(* CODESYS project Singla_Jagdamba_Rice_Final_28_02_20.project
   Title: Singla_Jagdamba_Rice_23_09_18
   Version: 0.0.0.0

Project tree, tasks and I/O mapping:
  MyController : TM218LDA40DRN, Schneider Electric, order no. TM218LDA40DRN, version 4.0.1.26
    application Application
      task MAST (cyclic, interval 20 ms, priority 15, watchdog 100 ms x 1) calls MainPOU
      function HiddenPOU [ST]
      global variables GVL
      program MainPOU [LD]
      function block fx1 [ST]
      function block fx2 [ST]
      function block CylOpenClose [ST]
    Embedded Functions
      IO : IO, Schneider Electric, version 4.0.1.26
          input  ES1 : BOOL  // ID0.I0
          input  ES2 : BOOL  // ID0.I1
          input  ES3 : BOOL  // ID0.I2
          input  ES4 : BOOL  // ID0.I3
          input  ES5 : BOOL  // ID0.I4
          input  ES6 : BOOL  // ID0.I5
          input  ES7 : BOOL  // ID0.I6
          input  ES8 : BOOL  // ID0.I7
          input  PS1 : BOOL  // ID0.I8
          input  PS2 : BOOL  // ID0.I9
          input  PS3 : BOOL  // ID0.I10
          input  PS4 : BOOL  // ID0.I11
          input  PS5 : BOOL  // ID0.I12
          input  PS6 : BOOL  // ID0.I13
          input  PS7 : BOOL  // ID0.I14
          input  PS8 : BOOL  // ID0.I15
          output qCylinder1 : BOOL  // QW0.Q0
          output qCylinder2 : BOOL  // QW0.Q1
          output qCylinder3 : BOOL  // QW0.Q2
          output qCylinder4 : BOOL  // QW0.Q3
          output qCylinder5 : BOOL  // QW0.Q4
          output qCylinder6 : BOOL  // QW0.Q5
          output qCylinder7 : BOOL  // QW0.Q6
          output qCylinder8 : BOOL  // QW0.Q7
          output qCylinder9 : BOOL  // QW0.Q8
          output qCylinder10 : BOOL  // QW0.Q9
          output qCylinder11 : BOOL  // QW0.Q10
          output qCylinder12 : BOOL  // QW0.Q11
          output qCylinder13 : BOOL  // QW0.Q12
          output qCylinder14 : BOOL  // QW0.Q13
          unmapped channels: ID0, QW0
      HSC : HSC, Schneider Electric, version 4.0.1.26
    Serial Line 1
      SoMachine_Network_Manager : SoMachine-Network Manager, Schneider Electric, version 4.0.0.2
    Serial Line 2
      Modbus_Manager : Modbus Manager, Schneider Electric, version 4.0.0.2
*)

// MyController/Application/GVL
VAR_GLOBAL
	
	k1TopCylClose: BOOL;
	k2TopCylClose: BOOL;
	k3TopCylClose: BOOL;
	k4TopCylClose: BOOL;
	k5TopCylClose: BOOL;
	k6TopCylClose: BOOL;
	
	manualOpenCyl1 AT %MX608.0: BOOL;
	manualOpenCyl2 AT %MX608.1: BOOL;
	manualOpenCyl3 AT %MX608.2: BOOL;
	manualOpenCyl4 AT %MX608.3: BOOL;
	manualOpenCyl5 AT %MX608.4: BOOL;
	manualOpenCyl6 AT %MX608.5: BOOL;
	manualOpenCyl7 AT %MX608.6: BOOL;
	manualOpenCyl8 AT %MX608.7: BOOL;
	manualOpenCyl9 AT %MX609.0: BOOL;
	manualOpenCyl10 AT %MX609.1: BOOL;
	manualOpenCyl11 AT %MX617.0: BOOL;
	manualOpenCyl12 AT %MX617.1: BOOL;
	manualOpenCyl13 AT %MX617.2: BOOL;
	manualOpenCyl14 AT %MX617.3: BOOL;
	
	manualCloseCyl1 AT %MX609.2: BOOL;
	manualCloseCyl2 AT %MX609.3: BOOL;
	manualCloseCyl3 AT %MX609.4: BOOL;
	manualCloseCyl4 AT %MX609.5: BOOL;
	manualCloseCyl5 AT %MX609.6: BOOL;
	manualCloseCyl6 AT %MX609.7: BOOL;
	manualCloseCyl7 AT %MX610.0: BOOL;
	manualCloseCyl8 AT %MX610.1: BOOL;
	manualCloseCyl9 AT %MX610.2: BOOL;
	manualCloseCyl10 AT %MX610.3: BOOL;
	manualCloseCyl11 AT %MX617.4: BOOL;
	manualCloseCyl12 AT %MX617.5: BOOL;
	manualCloseCyl13 AT %MX617.6: BOOL;
	manualCloseCyl14 AT %MX617.7: BOOL;
	
	
	openCyl1 AT %MX603.2: BOOL;
	openCyl2 AT %MX603.3: BOOL;
	openCyl3 AT %MX603.4: BOOL;
	openCyl4 AT %MX603.5: BOOL;
	openCyl5 AT %MX603.6: BOOL;
	openCyl6 AT %MX603.7: BOOL;
	openCyl7 AT %MX604.0: BOOL;
	openCyl8 AT %MX604.1: BOOL;
	openCyl9 AT %MX604.2: BOOL;
	openCyl10 AT %MX604.3: BOOL;
	openCyl11 AT %MX618.0: BOOL;
	openCyl12 AT %MX618.1: BOOL;
	openCyl13 AT %MX618.2: BOOL;
	openCyl14 AT %MX618.3: BOOL;
	
	k1CycleStart AT %MX606.0: BOOL;
	k2CycleStart AT %MX606.1: BOOL;
	k3CycleStart AT %MX606.2: BOOL;
	k4CycleStart AT %MX606.3: BOOL;
	k5CycleStart AT %MX618.4: BOOL;
	k6CycleStart AT %MX618.5: BOOL;
	p1CycleStart AT %MX606.4: BOOL;
	p2CycleStart AT %MX606.5: BOOL;
	
	k1CycleStop AT %MX606.6: BOOL;
	k2CycleStop AT %MX606.7: BOOL;
	k3CycleStop AT %MX607.0: BOOL;
	k4CycleStop AT %MX607.1: BOOL;
	k5CycleStop AT %MX618.6: BOOL;
	k6CycleStop AT %MX618.7: BOOL;
	p1CycleStop AT %MX607.2: BOOL;
	p2CycleStop AT %MX607.3: BOOL;
	
	k1Start AT %MX612.0: BOOL;
	k2Start AT %MX612.1: BOOL;
	k3Start AT %MX612.2: BOOL;
	k4Start AT %MX612.3: BOOL;
	k5Start AT %MX619.0: BOOL;
	k6Start AT %MX619.1: BOOL;
	p1Start AT %MX612.4: BOOL;
	p2Start AT %MX612.5: BOOL;

	k1CountComplete AT %MX612.6: BOOL;
	k2CountComplete AT %MX612.7: BOOL;
	k3CountComplete AT %MX613.0: BOOL;
	k4CountComplete AT %MX613.1: BOOL;
	k5CountComplete AT %MX619.2: BOOL;
	k6CountComplete AT %MX619.3: BOOL;
	p1CountComplete AT %MX613.2: BOOL;
	p2CountComplete AT %MX613.3: BOOL;
	
	k1PressureLow AT %MX613.4: BOOL;
	k2PressureLow AT %MX613.5: BOOL;
	k3PressureLow AT %MX613.6: BOOL;
	k4PressureLow AT %MX613.7: BOOL;
	k5PressureLow AT %MX619.4: BOOL;
	k6PressureLow AT %MX619.5: BOOL;
	p1PressureLow AT %MX614.0: BOOL;
	p2PressureLow AT %MX614.1: BOOL;
	
	k1Reset AT %MX616.0: BOOL;
	k2Reset AT %MX616.1: BOOL;
	k3Reset AT %MX616.2: BOOL;
	k4Reset AT %MX616.3: BOOL;
	k5Reset AT %MX619.6: BOOL;
	k6Reset AT %MX619.7: BOOL;
	p1Reset AT %MX616.4: BOOL;
	p2Reset AT %MX616.5: BOOL;
	
	k1ActCycleTime AT %MW122: INT; //in minutes
	k2ActCycleTime AT %MW123: INT;
	k3ActCycleTime AT %MW124: INT;
	k4ActCycleTime AT %MW125: INT;
	k5ActCycleTime AT %MW152: INT;
	k6ActCycleTime AT %MW153: INT;
	p1ActCycleTime AT %MW126: INT;
	p2ActCycleTime AT %MW127: INT;
	
	k1ActCount AT %MW128: INT;
	k2ActCount AT %MW129: INT;
	k3ActCount AT %MW130: INT;
	k4ActCount AT %MW131: INT;
	k5ActCount AT %MW150: INT;
	k6ActCount AT %MW151: INT;
	p1ActCount AT %MW132: INT;
	p2ActCount AT %MW133: INT;
	
END_VAR

VAR_GLOBAL RETAIN
	k1SetCount AT %MW100: INT := 15;
	k2SetCount AT %MW101: INT := 15;
	k3SetCount AT %MW102: INT := 15;
	k4SetCount AT %MW103: INT := 15;
	k5SetCount AT %MW148: INT := 15;
	k6SetCount AT %MW149: INT := 15;
	p1SetCount AT %MW104: INT := 5;
	p2SetCount AT %MW105: INT := 5;
	
	setTimeCylOpen1 AT %MW106: INT := 15; //in seconds
	setTimeCylOpen2 AT %MW107: INT := 15;
	setTimeCylOpen3 AT %MW108: INT := 15;
	setTimeCylOpen4 AT %MW109: INT := 15;
	setTimeCylOpen5 AT %MW110: INT := 15;
	setTimeCylOpen6 AT %MW111: INT := 15;
	setTimeCylOpen7 AT %MW112: INT := 15;
	setTimeCylOpen8 AT %MW113: INT := 15;
	setTimeCylOpen9 AT %MW114: INT := 15;
	setTimeCylOpen10 AT %MW115: INT := 15;
	setTimeCylOpen11 AT %MW144: INT := 15;
	setTimeCylOpen12 AT %MW145: INT := 15;
	setTimeCylOpen13 AT %MW146: INT := 15;
	setTimeCylOpen14 AT %MW147: INT := 15;
	
	
	k1SetCycleTime AT %MW116: INT := 15;
	k2SetCycleTime AT %MW117: INT := 15;
	k3SetCycleTime AT %MW118: INT := 15;
	k4SetCycleTime AT %MW119: INT := 15;
	k5SetCycleTime AT %MW142: INT := 15;
	k6SetCycleTime AT %MW143: INT := 15;
	p1SetCycleTime AT %MW120: INT := 15;
	p2SetCycleTime AT %MW121: INT := 15;
	
	k1SetCloseCount AT %MW134: INT := 2;
	k2SetCloseCount AT %MW135: INT := 2;
	k3SetCloseCount AT %MW136: INT := 2;
	k4SetCloseCount AT %MW137: INT := 2;
	k5SetCloseCount AT %MW140: INT := 2;
	k6SetCloseCount AT %MW141: INT := 2;
	p1SetCloseCount AT %MW138: INT;
	p2SetCloseCount AT %MW139: INT;
	
	k1ManualOverride AT %MX600.0: BOOL;
	k2ManualOverride AT %MX600.1: BOOL;
	k3ManualOverride AT %MX600.2: BOOL;
	k4ManualOverride AT %MX600.3: BOOL;
	k5ManualOverride AT %MX620.0: BOOL;
	k6ManualOverride AT %MX620.1: BOOL;
	p1ManualOverride AT %MX600.4: BOOL;
	p2ManualOverride AT %MX600.5: BOOL;

END_VAR

// MyController/Application/MainPOU
PROGRAM MainPOU
VAR

	Kacchi_1: fx1;
	Kacchi_1_Count: fx2;
	Kacchi_2: fx1;
	Kacchi_2_Count: fx2;
	Kacchi_3_Count: fx2;
	Kacchi_3: fx1;
	Kacchi_4: fx1;
	Kacchi_4_Count: fx2;
	Pakki_1: fx1;
	Pakki_1_Count: fx2;
	Pakki_2: fx1;
	Pakki_2_Count: fx2;
	
	
	k2BottomCmd: BOOL;
	k1BottomCmd: BOOL;
	k3BottomCmd: BOOL;
	k4BottomCmd: BOOL;
	p1BottomCmd: BOOL;
	p2BottomCmd: BOOL;
	
	CylOpenClose_0: CylOpenClose;
	CylOpenClose_1: CylOpenClose;
	CylOpenClose_2: CylOpenClose;
	CylOpenClose_3: CylOpenClose;
	CylOpenClose_4: CylOpenClose;
	CylOpenClose_5: CylOpenClose;
	CylOpenClose_6: CylOpenClose;
	CylOpenClose_7: CylOpenClose;
	CylOpenClose_8: CylOpenClose;
	CylOpenClose_9: CylOpenClose;
	p2Stop: BOOL;
	k4Stop: BOOL;
	p1Stop: BOOL;
	k3Stop: BOOL;
	k2Stop: BOOL;
	k1Stop: BOOL;
	
	R_TRIG_0: R_TRIG;
	R_TRIG_1: R_TRIG;
	R_TRIG_2: R_TRIG;
	R_TRIG_3: R_TRIG;
	R_TRIG_4: R_TRIG;
	R_TRIG_5: R_TRIG;
	R_TRIG_6: R_TRIG;
	R_TRIG_7: R_TRIG;
	R_TRIG_8: R_TRIG;
	R_TRIG_9: R_TRIG;
	RS_6: RS;
	k6Stop: BOOL;
	R_TRIG_15: R_TRIG;
	R_TRIG_16: R_TRIG;
	RS_7: RS;
	Kacchi_5: fx1;
	k5BottomCmd: BOOL;
	Kacchi_5_Count: fx2;
	k5Stop: BOOL;
	Kacchi_6: fx1;
	k6BottomCmd: BOOL;
	Kacchi_6_Count: fx2;
	CylOpenClose_10: CylOpenClose;
	R_TRIG_10: R_TRIG;
	CylOpenClose_11: CylOpenClose;
	CylOpenClose_12: CylOpenClose;
	R_TRIG_12: R_TRIG;
	CylOpenClose_13: CylOpenClose;
END_VAR

VAR RETAIN
	RS_0: RS;
	RS_1: RS;
	RS_2: RS;
	RS_3: RS;
	RS_4: RS;
	RS_5: RS;
END_VAR
VAR // added by the converter: edge detectors and wires of the graphical bodies
    _w1, _w2 : BOOL;
END_VAR

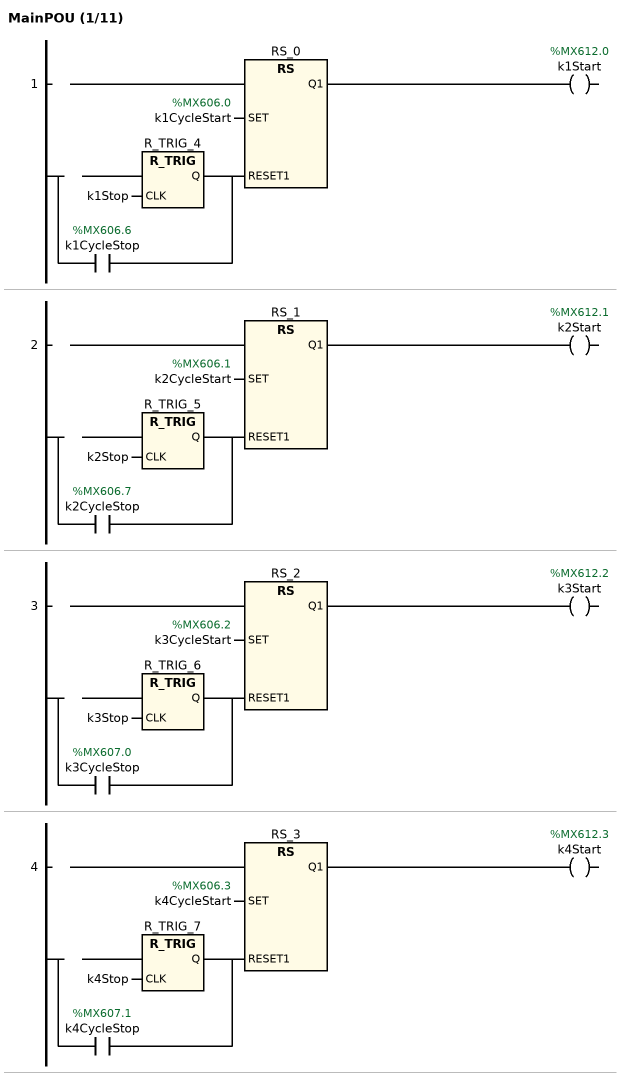
// NETWORK 1
//   k1CycleStart: AT %MX606.0
//   k1CycleStop: AT %MX606.6
//   k1Start: AT %MX612.0
R_TRIG_4(CLK := k1Stop); // R_TRIG
RS_0(SET := k1CycleStart, RESET1 := R_TRIG_4.Q OR k1CycleStop); // RS
k1Start := RS_0.Q1;

// NETWORK 2
//   k2CycleStart: AT %MX606.1
//   k2CycleStop: AT %MX606.7
//   k2Start: AT %MX612.1
R_TRIG_5(CLK := k2Stop); // R_TRIG
RS_1(SET := k2CycleStart, RESET1 := R_TRIG_5.Q OR k2CycleStop); // RS
k2Start := RS_1.Q1;

// NETWORK 3
//   k3CycleStart: AT %MX606.2
//   k3CycleStop: AT %MX607.0
//   k3Start: AT %MX612.2
R_TRIG_6(CLK := k3Stop); // R_TRIG
RS_2(SET := k3CycleStart, RESET1 := R_TRIG_6.Q OR k3CycleStop); // RS
k3Start := RS_2.Q1;

// NETWORK 4
//   k4CycleStart: AT %MX606.3
//   k4CycleStop: AT %MX607.1
//   k4Start: AT %MX612.3
R_TRIG_7(CLK := k4Stop); // R_TRIG
RS_3(SET := k4CycleStart, RESET1 := R_TRIG_7.Q OR k4CycleStop); // RS
k4Start := RS_3.Q1;

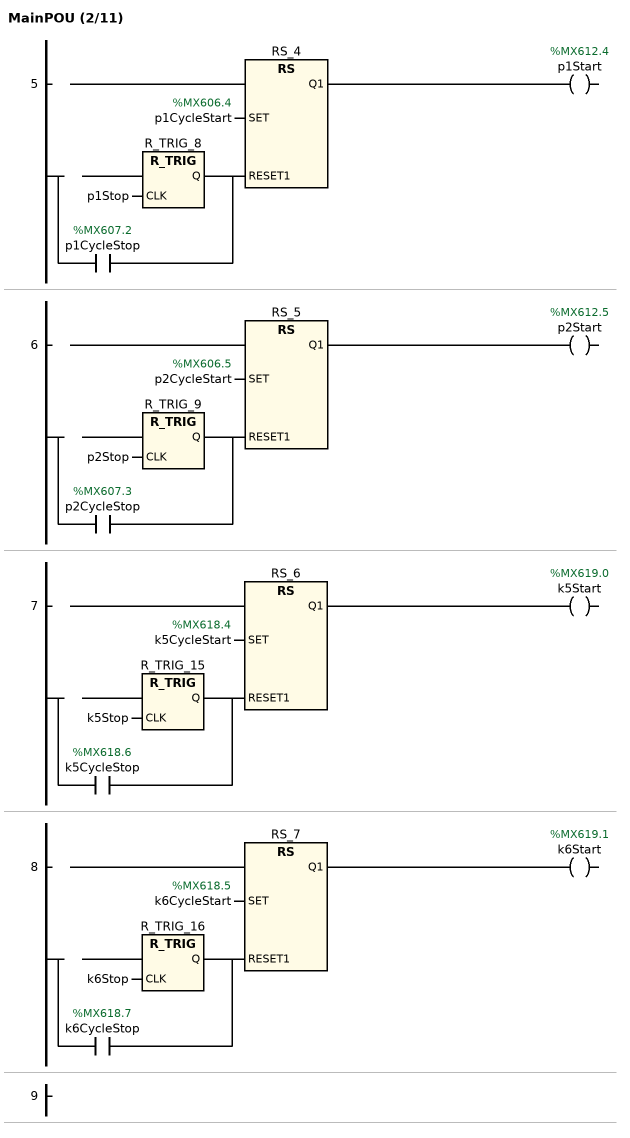
// NETWORK 5
//   p1CycleStart: AT %MX606.4
//   p1CycleStop: AT %MX607.2
//   p1Start: AT %MX612.4
R_TRIG_8(CLK := p1Stop); // R_TRIG
RS_4(SET := p1CycleStart, RESET1 := R_TRIG_8.Q OR p1CycleStop); // RS
p1Start := RS_4.Q1;

// NETWORK 6
//   p2CycleStart: AT %MX606.5
//   p2CycleStop: AT %MX607.3
//   p2Start: AT %MX612.5
R_TRIG_9(CLK := p2Stop); // R_TRIG
RS_5(SET := p2CycleStart, RESET1 := R_TRIG_9.Q OR p2CycleStop); // RS
p2Start := RS_5.Q1;

// NETWORK 7
//   k5CycleStart: AT %MX618.4
//   k5CycleStop: AT %MX618.6
//   k5Start: AT %MX619.0
R_TRIG_15(CLK := k5Stop); // R_TRIG
RS_6(SET := k5CycleStart, RESET1 := R_TRIG_15.Q OR k5CycleStop); // RS
k5Start := RS_6.Q1;

// NETWORK 8
//   k6CycleStart: AT %MX618.5
//   k6CycleStop: AT %MX618.7
//   k6Start: AT %MX619.1
R_TRIG_16(CLK := k6Stop); // R_TRIG
RS_7(SET := k6CycleStart, RESET1 := R_TRIG_16.Q OR k6CycleStop); // RS
k6Start := RS_7.Q1;

// NETWORK 9

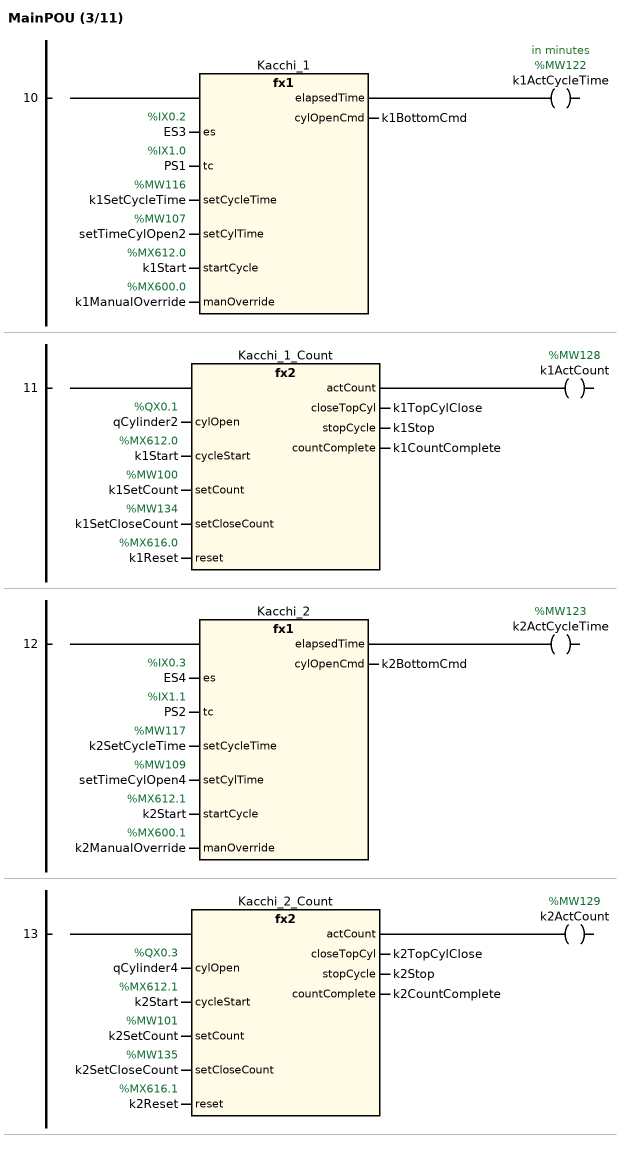
// NETWORK 10
//   ES3: IO : | AT %IX0.2
//   PS1: IO : | AT %IX1.0
//   k1SetCycleTime: AT %MW116
//   setTimeCylOpen2: AT %MW107
//   k1Start: AT %MX612.0
//   k1ManualOverride: AT %MX600.0
//   k1ActCycleTime: in minutes | AT %MW122
Kacchi_1(
    es := ES3,
    tc := PS1,
    setCycleTime := k1SetCycleTime,
    setCylTime := setTimeCylOpen2,
    startCycle := k1Start,
    manOverride := k1ManualOverride,
    cylOpenCmd => k1BottomCmd); // fx1
k1ActCycleTime := Kacchi_1.elapsedTime;

// NETWORK 11
//   qCylinder2: IO : | AT %QX0.1
//   k1Start: AT %MX612.0
//   k1SetCount: AT %MW100
//   k1SetCloseCount: AT %MW134
//   k1Reset: AT %MX616.0
//   k1CountComplete: AT %MX612.6
//   k1ActCount: AT %MW128
Kacchi_1_Count(
    cylOpen := qCylinder2,
    cycleStart := k1Start,
    setCount := k1SetCount,
    setCloseCount := k1SetCloseCount,
    reset := k1Reset,
    closeTopCyl => k1TopCylClose,
    stopCycle => k1Stop,
    countComplete => k1CountComplete); // fx2
k1ActCount := Kacchi_1_Count.actCount;

// NETWORK 12
//   ES4: IO : | AT %IX0.3
//   PS2: IO : | AT %IX1.1
//   k2SetCycleTime: AT %MW117
//   setTimeCylOpen4: AT %MW109
//   k2Start: AT %MX612.1
//   k2ManualOverride: AT %MX600.1
//   k2ActCycleTime: AT %MW123
Kacchi_2(
    es := ES4,
    tc := PS2,
    setCycleTime := k2SetCycleTime,
    setCylTime := setTimeCylOpen4,
    startCycle := k2Start,
    manOverride := k2ManualOverride,
    cylOpenCmd => k2BottomCmd); // fx1
k2ActCycleTime := Kacchi_2.elapsedTime;

// NETWORK 13
//   qCylinder4: IO : | AT %QX0.3
//   k2Start: AT %MX612.1
//   k2SetCount: AT %MW101
//   k2SetCloseCount: AT %MW135
//   k2Reset: AT %MX616.1
//   k2CountComplete: AT %MX612.7
//   k2ActCount: AT %MW129
Kacchi_2_Count(
    cylOpen := qCylinder4,
    cycleStart := k2Start,
    setCount := k2SetCount,
    setCloseCount := k2SetCloseCount,
    reset := k2Reset,
    closeTopCyl => k2TopCylClose,
    stopCycle => k2Stop,
    countComplete => k2CountComplete); // fx2
k2ActCount := Kacchi_2_Count.actCount;

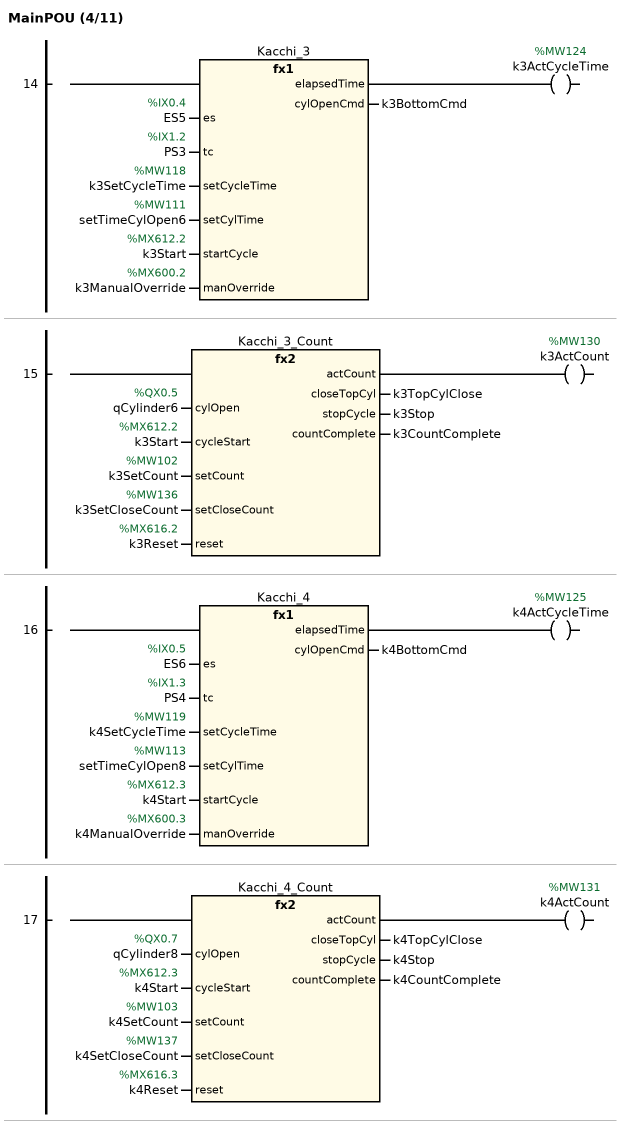
// NETWORK 14
//   ES5: IO : | AT %IX0.4
//   PS3: IO : | AT %IX1.2
//   k3SetCycleTime: AT %MW118
//   setTimeCylOpen6: AT %MW111
//   k3Start: AT %MX612.2
//   k3ManualOverride: AT %MX600.2
//   k3ActCycleTime: AT %MW124
Kacchi_3(
    es := ES5,
    tc := PS3,
    setCycleTime := k3SetCycleTime,
    setCylTime := setTimeCylOpen6,
    startCycle := k3Start,
    manOverride := k3ManualOverride,
    cylOpenCmd => k3BottomCmd); // fx1
k3ActCycleTime := Kacchi_3.elapsedTime;

// NETWORK 15
//   qCylinder6: IO : | AT %QX0.5
//   k3Start: AT %MX612.2
//   k3SetCount: AT %MW102
//   k3SetCloseCount: AT %MW136
//   k3Reset: AT %MX616.2
//   k3CountComplete: AT %MX613.0
//   k3ActCount: AT %MW130
Kacchi_3_Count(
    cylOpen := qCylinder6,
    cycleStart := k3Start,
    setCount := k3SetCount,
    setCloseCount := k3SetCloseCount,
    reset := k3Reset,
    closeTopCyl => k3TopCylClose,
    stopCycle => k3Stop,
    countComplete => k3CountComplete); // fx2
k3ActCount := Kacchi_3_Count.actCount;

// NETWORK 16
//   ES6: IO : | AT %IX0.5
//   PS4: IO : | AT %IX1.3
//   k4SetCycleTime: AT %MW119
//   setTimeCylOpen8: AT %MW113
//   k4Start: AT %MX612.3
//   k4ManualOverride: AT %MX600.3
//   k4ActCycleTime: AT %MW125
Kacchi_4(
    es := ES6,
    tc := PS4,
    setCycleTime := k4SetCycleTime,
    setCylTime := setTimeCylOpen8,
    startCycle := k4Start,
    manOverride := k4ManualOverride,
    cylOpenCmd => k4BottomCmd); // fx1
k4ActCycleTime := Kacchi_4.elapsedTime;

// NETWORK 17
//   qCylinder8: IO : | AT %QX0.7
//   k4Start: AT %MX612.3
//   k4SetCount: AT %MW103
//   k4SetCloseCount: AT %MW137
//   k4Reset: AT %MX616.3
//   k4CountComplete: AT %MX613.1
//   k4ActCount: AT %MW131
Kacchi_4_Count(
    cylOpen := qCylinder8,
    cycleStart := k4Start,
    setCount := k4SetCount,
    setCloseCount := k4SetCloseCount,
    reset := k4Reset,
    closeTopCyl => k4TopCylClose,
    stopCycle => k4Stop,
    countComplete => k4CountComplete); // fx2
k4ActCount := Kacchi_4_Count.actCount;

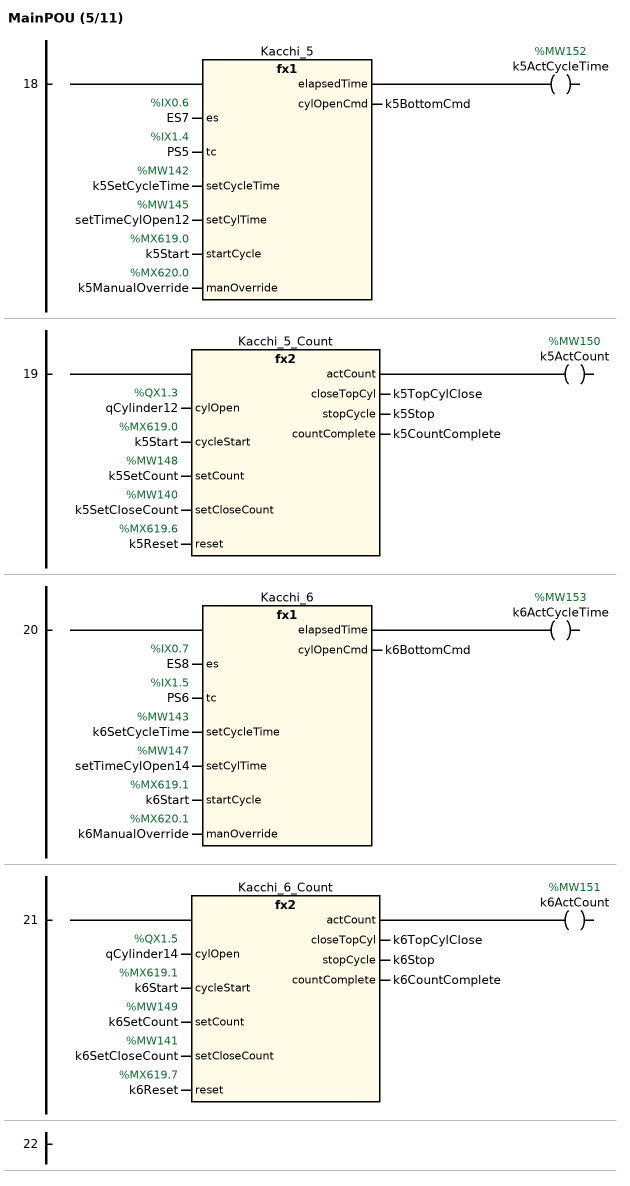
// NETWORK 18
//   ES7: IO : | AT %IX0.6
//   PS5: IO : | AT %IX1.4
//   k5SetCycleTime: AT %MW142
//   setTimeCylOpen12: AT %MW145
//   k5Start: AT %MX619.0
//   k5ManualOverride: AT %MX620.0
//   k5ActCycleTime: AT %MW152
Kacchi_5(
    es := ES7,
    tc := PS5,
    setCycleTime := k5SetCycleTime,
    setCylTime := setTimeCylOpen12,
    startCycle := k5Start,
    manOverride := k5ManualOverride,
    cylOpenCmd => k5BottomCmd); // fx1
k5ActCycleTime := Kacchi_5.elapsedTime;

// NETWORK 19
//   qCylinder12: IO : | AT %QX1.3
//   k5Start: AT %MX619.0
//   k5SetCount: AT %MW148
//   k5SetCloseCount: AT %MW140
//   k5Reset: AT %MX619.6
//   k5CountComplete: AT %MX619.2
//   k5ActCount: AT %MW150
Kacchi_5_Count(
    cylOpen := qCylinder12,
    cycleStart := k5Start,
    setCount := k5SetCount,
    setCloseCount := k5SetCloseCount,
    reset := k5Reset,
    closeTopCyl => k5TopCylClose,
    stopCycle => k5Stop,
    countComplete => k5CountComplete); // fx2
k5ActCount := Kacchi_5_Count.actCount;

// NETWORK 20
//   ES8: IO : | AT %IX0.7
//   PS6: IO : | AT %IX1.5
//   k6SetCycleTime: AT %MW143
//   setTimeCylOpen14: AT %MW147
//   k6Start: AT %MX619.1
//   k6ManualOverride: AT %MX620.1
//   k6ActCycleTime: AT %MW153
Kacchi_6(
    es := ES8,
    tc := PS6,
    setCycleTime := k6SetCycleTime,
    setCylTime := setTimeCylOpen14,
    startCycle := k6Start,
    manOverride := k6ManualOverride,
    cylOpenCmd => k6BottomCmd); // fx1
k6ActCycleTime := Kacchi_6.elapsedTime;

// NETWORK 21
//   qCylinder14: IO : | AT %QX1.5
//   k6Start: AT %MX619.1
//   k6SetCount: AT %MW149
//   k6SetCloseCount: AT %MW141
//   k6Reset: AT %MX619.7
//   k6CountComplete: AT %MX619.3
//   k6ActCount: AT %MW151
Kacchi_6_Count(
    cylOpen := qCylinder14,
    cycleStart := k6Start,
    setCount := k6SetCount,
    setCloseCount := k6SetCloseCount,
    reset := k6Reset,
    closeTopCyl => k6TopCylClose,
    stopCycle => k6Stop,
    countComplete => k6CountComplete); // fx2
k6ActCount := Kacchi_6_Count.actCount;

// NETWORK 22

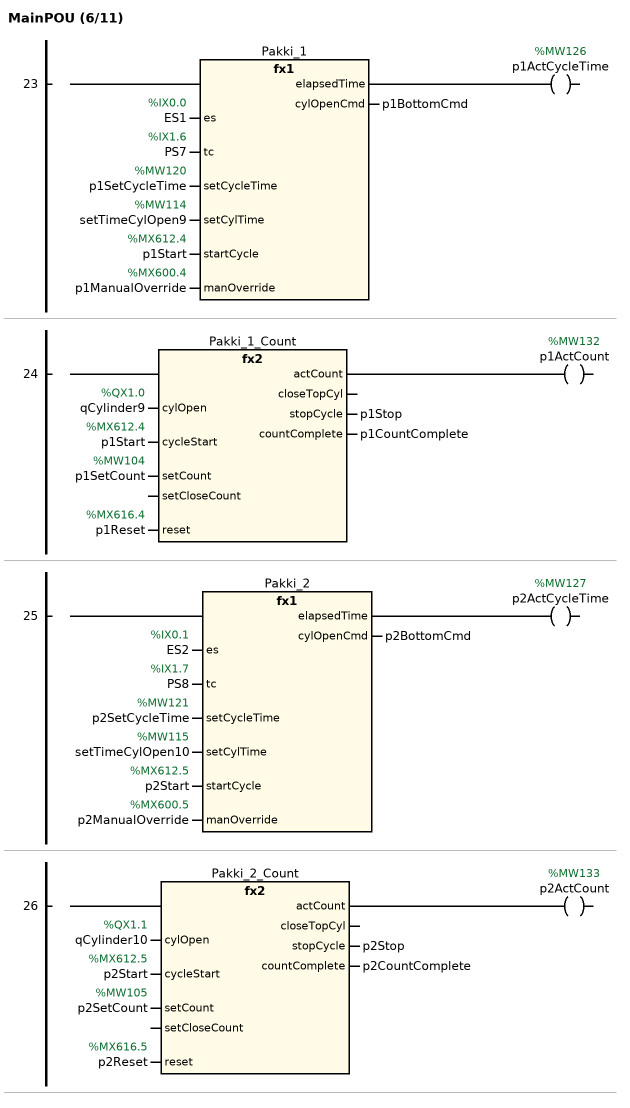
// NETWORK 23
//   ES1: IO : Fast Input | AT %IX0.0
//   PS7: IO : | AT %IX1.6
//   p1SetCycleTime: AT %MW120
//   setTimeCylOpen9: AT %MW114
//   p1Start: AT %MX612.4
//   p1ManualOverride: AT %MX600.4
//   p1ActCycleTime: AT %MW126
Pakki_1(
    es := ES1,
    tc := PS7,
    setCycleTime := p1SetCycleTime,
    setCylTime := setTimeCylOpen9,
    startCycle := p1Start,
    manOverride := p1ManualOverride,
    cylOpenCmd => p1BottomCmd); // fx1
p1ActCycleTime := Pakki_1.elapsedTime;

// NETWORK 24
//   qCylinder9: IO : | AT %QX1.0
//   p1Start: AT %MX612.4
//   p1SetCount: AT %MW104
//   p1Reset: AT %MX616.4
//   p1CountComplete: AT %MX613.2
//   p1ActCount: AT %MW132
Pakki_1_Count(
    cylOpen := qCylinder9,
    cycleStart := p1Start,
    setCount := p1SetCount,
    reset := p1Reset,
    stopCycle => p1Stop,
    countComplete => p1CountComplete); // fx2
p1ActCount := Pakki_1_Count.actCount;

// NETWORK 25
//   ES2: IO : Fast Input | AT %IX0.1
//   PS8: IO : | AT %IX1.7
//   p2SetCycleTime: AT %MW121
//   setTimeCylOpen10: AT %MW115
//   p2Start: AT %MX612.5
//   p2ManualOverride: AT %MX600.5
//   p2ActCycleTime: AT %MW127
Pakki_2(
    es := ES2,
    tc := PS8,
    setCycleTime := p2SetCycleTime,
    setCylTime := setTimeCylOpen10,
    startCycle := p2Start,
    manOverride := p2ManualOverride,
    cylOpenCmd => p2BottomCmd); // fx1
p2ActCycleTime := Pakki_2.elapsedTime;

// NETWORK 26
//   qCylinder10: IO : | AT %QX1.1
//   p2Start: AT %MX612.5
//   p2SetCount: AT %MW105
//   p2Reset: AT %MX616.5
//   p2CountComplete: AT %MX613.3
//   p2ActCount: AT %MW133
Pakki_2_Count(
    cylOpen := qCylinder10,
    cycleStart := p2Start,
    setCount := p2SetCount,
    reset := p2Reset,
    stopCycle => p2Stop,
    countComplete => p2CountComplete); // fx2
p2ActCount := Pakki_2_Count.actCount;

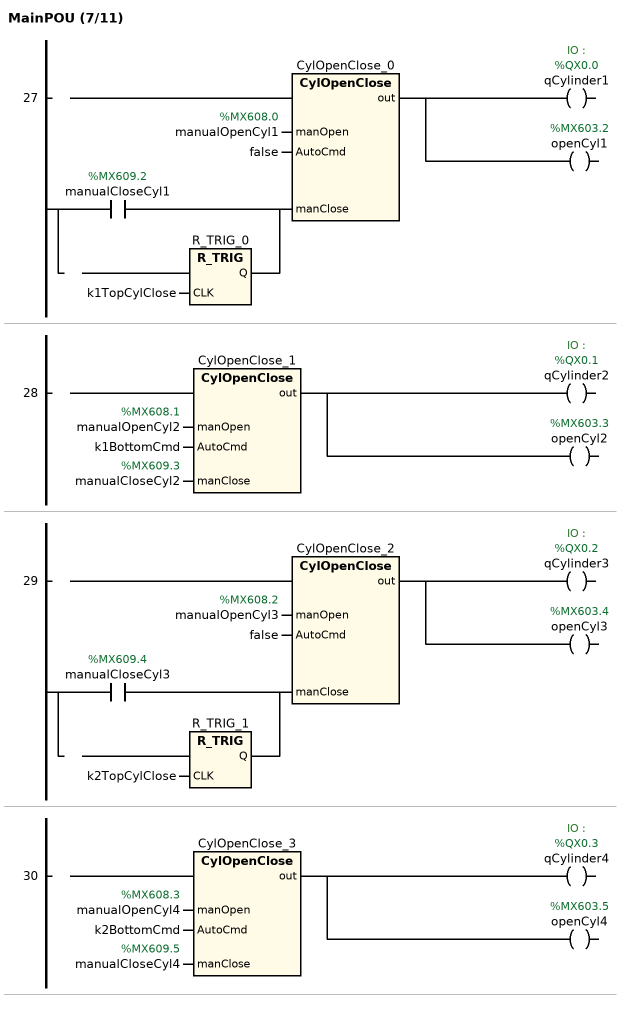
// NETWORK 27
//   manualOpenCyl1: AT %MX608.0
//   manualCloseCyl1: AT %MX609.2
//   qCylinder1: IO : | AT %QX0.0
//   openCyl1: AT %MX603.2
R_TRIG_0(CLK := k1TopCylClose); // R_TRIG
CylOpenClose_0(manOpen := manualOpenCyl1, AutoCmd := false, manClose := manualCloseCyl1 OR R_TRIG_0.Q); // CylOpenClose
qCylinder1 := CylOpenClose_0.out;
openCyl1 := CylOpenClose_0.out;

// NETWORK 28
//   manualOpenCyl2: AT %MX608.1
//   manualCloseCyl2: AT %MX609.3
//   qCylinder2: IO : | AT %QX0.1
//   openCyl2: AT %MX603.3
CylOpenClose_1(manOpen := manualOpenCyl2, AutoCmd := k1BottomCmd, manClose := manualCloseCyl2); // CylOpenClose
qCylinder2 := CylOpenClose_1.out;
openCyl2 := CylOpenClose_1.out;

// NETWORK 29
//   manualOpenCyl3: AT %MX608.2
//   manualCloseCyl3: AT %MX609.4
//   qCylinder3: IO : | AT %QX0.2
//   openCyl3: AT %MX603.4
R_TRIG_1(CLK := k2TopCylClose); // R_TRIG
CylOpenClose_2(manOpen := manualOpenCyl3, AutoCmd := false, manClose := manualCloseCyl3 OR R_TRIG_1.Q); // CylOpenClose
qCylinder3 := CylOpenClose_2.out;
openCyl3 := CylOpenClose_2.out;

// NETWORK 30
//   manualOpenCyl4: AT %MX608.3
//   manualCloseCyl4: AT %MX609.5
//   qCylinder4: IO : | AT %QX0.3
//   openCyl4: AT %MX603.5
CylOpenClose_3(manOpen := manualOpenCyl4, AutoCmd := k2BottomCmd, manClose := manualCloseCyl4); // CylOpenClose
qCylinder4 := CylOpenClose_3.out;
openCyl4 := CylOpenClose_3.out;

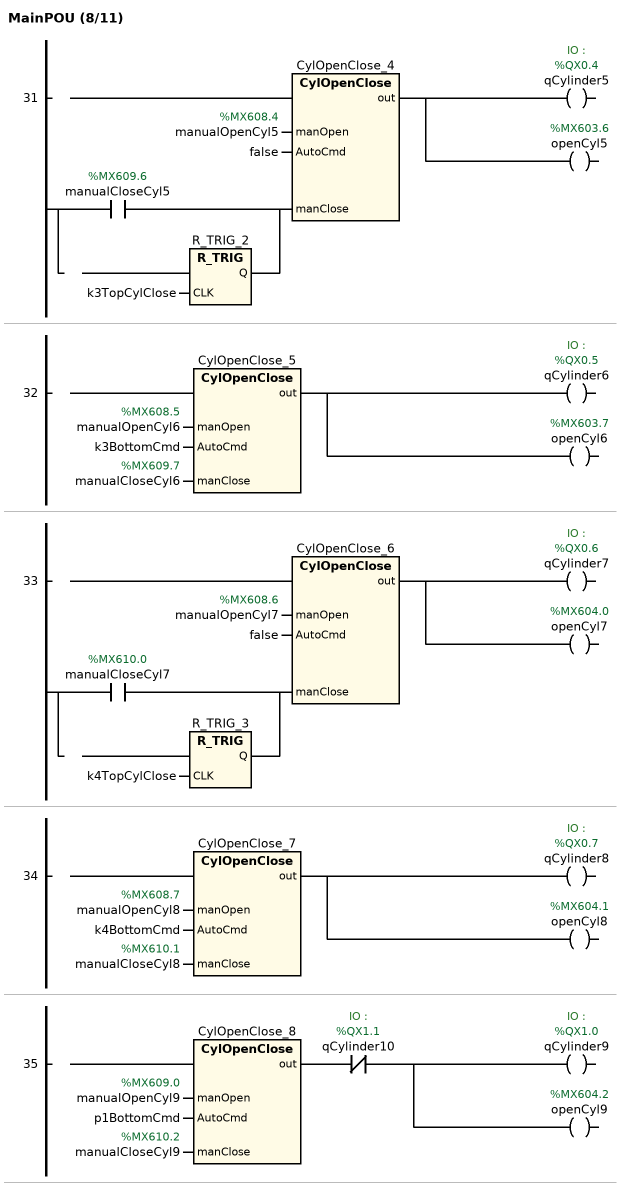
// NETWORK 31
//   manualOpenCyl5: AT %MX608.4
//   manualCloseCyl5: AT %MX609.6
//   qCylinder5: IO : | AT %QX0.4
//   openCyl5: AT %MX603.6
R_TRIG_2(CLK := k3TopCylClose); // R_TRIG
CylOpenClose_4(manOpen := manualOpenCyl5, AutoCmd := false, manClose := manualCloseCyl5 OR R_TRIG_2.Q); // CylOpenClose
qCylinder5 := CylOpenClose_4.out;
openCyl5 := CylOpenClose_4.out;

// NETWORK 32
//   manualOpenCyl6: AT %MX608.5
//   manualCloseCyl6: AT %MX609.7
//   qCylinder6: IO : | AT %QX0.5
//   openCyl6: AT %MX603.7
CylOpenClose_5(manOpen := manualOpenCyl6, AutoCmd := k3BottomCmd, manClose := manualCloseCyl6); // CylOpenClose
qCylinder6 := CylOpenClose_5.out;
openCyl6 := CylOpenClose_5.out;

// NETWORK 33
//   manualOpenCyl7: AT %MX608.6
//   manualCloseCyl7: AT %MX610.0
//   qCylinder7: IO : | AT %QX0.6
//   openCyl7: AT %MX604.0
R_TRIG_3(CLK := k4TopCylClose); // R_TRIG
CylOpenClose_6(manOpen := manualOpenCyl7, AutoCmd := false, manClose := manualCloseCyl7 OR R_TRIG_3.Q); // CylOpenClose
qCylinder7 := CylOpenClose_6.out;
openCyl7 := CylOpenClose_6.out;

// NETWORK 34
//   manualOpenCyl8: AT %MX608.7
//   manualCloseCyl8: AT %MX610.1
//   qCylinder8: IO : | AT %QX0.7
//   openCyl8: AT %MX604.1
CylOpenClose_7(manOpen := manualOpenCyl8, AutoCmd := k4BottomCmd, manClose := manualCloseCyl8); // CylOpenClose
qCylinder8 := CylOpenClose_7.out;
openCyl8 := CylOpenClose_7.out;

// NETWORK 35
//   manualOpenCyl9: AT %MX609.0
//   manualCloseCyl9: AT %MX610.2
//   qCylinder10: IO : | AT %QX1.1
//   qCylinder9: IO : | AT %QX1.0
//   openCyl9: AT %MX604.2
CylOpenClose_8(manOpen := manualOpenCyl9, AutoCmd := p1BottomCmd, manClose := manualCloseCyl9); // CylOpenClose
_w1 := CylOpenClose_8.out AND NOT qCylinder10;
qCylinder9 := _w1;
openCyl9 := _w1;

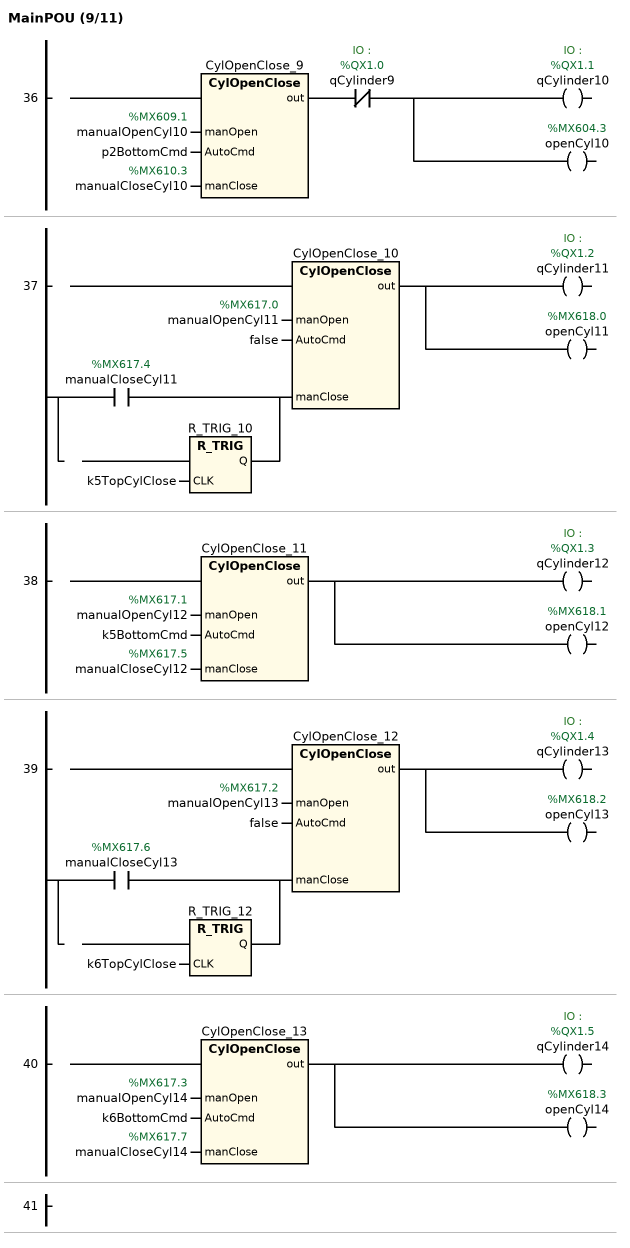
// NETWORK 36
//   manualOpenCyl10: AT %MX609.1
//   manualCloseCyl10: AT %MX610.3
//   qCylinder9: IO : | AT %QX1.0
//   qCylinder10: IO : | AT %QX1.1
//   openCyl10: AT %MX604.3
CylOpenClose_9(manOpen := manualOpenCyl10, AutoCmd := p2BottomCmd, manClose := manualCloseCyl10); // CylOpenClose
_w2 := CylOpenClose_9.out AND NOT qCylinder9;
qCylinder10 := _w2;
openCyl10 := _w2;

// NETWORK 37
//   manualOpenCyl11: AT %MX617.0
//   manualCloseCyl11: AT %MX617.4
//   qCylinder11: IO : | AT %QX1.2
//   openCyl11: AT %MX618.0
R_TRIG_10(CLK := k5TopCylClose); // R_TRIG
CylOpenClose_10(manOpen := manualOpenCyl11, AutoCmd := false, manClose := manualCloseCyl11 OR R_TRIG_10.Q); // CylOpenClose
qCylinder11 := CylOpenClose_10.out;
openCyl11 := CylOpenClose_10.out;

// NETWORK 38
//   manualOpenCyl12: AT %MX617.1
//   manualCloseCyl12: AT %MX617.5
//   qCylinder12: IO : | AT %QX1.3
//   openCyl12: AT %MX618.1
CylOpenClose_11(manOpen := manualOpenCyl12, AutoCmd := k5BottomCmd, manClose := manualCloseCyl12); // CylOpenClose
qCylinder12 := CylOpenClose_11.out;
openCyl12 := CylOpenClose_11.out;

// NETWORK 39
//   manualOpenCyl13: AT %MX617.2
//   manualCloseCyl13: AT %MX617.6
//   qCylinder13: IO : | AT %QX1.4
//   openCyl13: AT %MX618.2
R_TRIG_12(CLK := k6TopCylClose); // R_TRIG
CylOpenClose_12(manOpen := manualOpenCyl13, AutoCmd := false, manClose := manualCloseCyl13 OR R_TRIG_12.Q); // CylOpenClose
qCylinder13 := CylOpenClose_12.out;
openCyl13 := CylOpenClose_12.out;

// NETWORK 40
//   manualOpenCyl14: AT %MX617.3
//   manualCloseCyl14: AT %MX617.7
//   qCylinder14: IO : | AT %QX1.5
//   openCyl14: AT %MX618.3
CylOpenClose_13(manOpen := manualOpenCyl14, AutoCmd := k6BottomCmd, manClose := manualCloseCyl14); // CylOpenClose
qCylinder14 := CylOpenClose_13.out;
openCyl14 := CylOpenClose_13.out;

// NETWORK 41

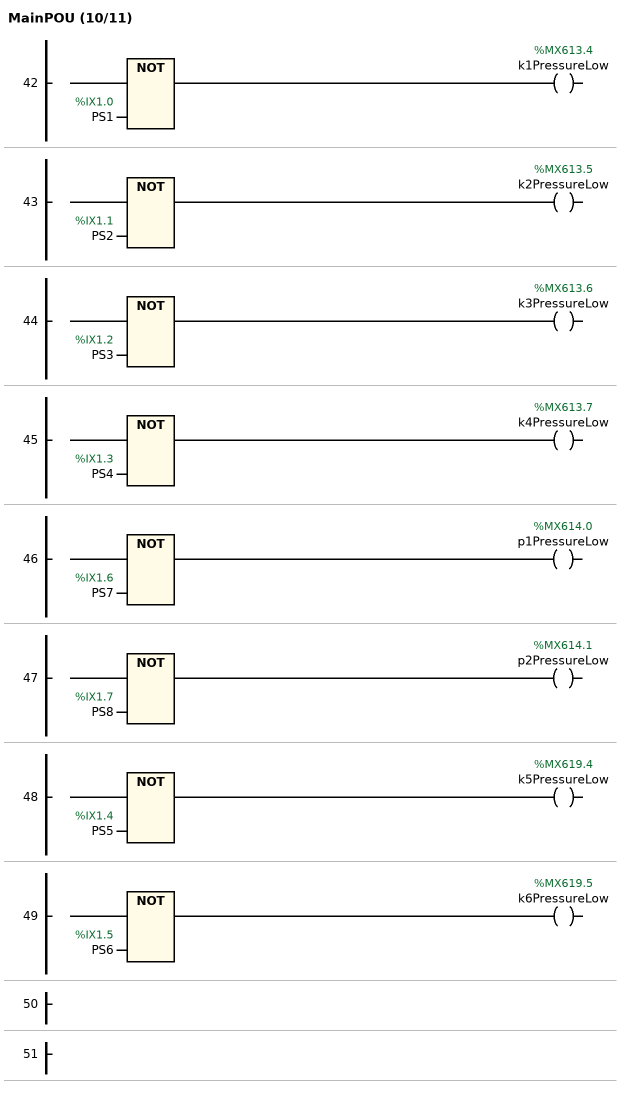
// NETWORK 42
//   PS1: IO : | AT %IX1.0
//   k1PressureLow: AT %MX613.4
k1PressureLow := NOT PS1;

// NETWORK 43
//   PS2: IO : | AT %IX1.1
//   k2PressureLow: AT %MX613.5
k2PressureLow := NOT PS2;

// NETWORK 44
//   PS3: IO : | AT %IX1.2
//   k3PressureLow: AT %MX613.6
k3PressureLow := NOT PS3;

// NETWORK 45
//   PS4: IO : | AT %IX1.3
//   k4PressureLow: AT %MX613.7
k4PressureLow := NOT PS4;

// NETWORK 46
//   PS7: IO : | AT %IX1.6
//   p1PressureLow: AT %MX614.0
p1PressureLow := NOT PS7;

// NETWORK 47
//   PS8: IO : | AT %IX1.7
//   p2PressureLow: AT %MX614.1
p2PressureLow := NOT PS8;

// NETWORK 48
//   PS5: IO : | AT %IX1.4
//   k5PressureLow: AT %MX619.4
k5PressureLow := NOT PS5;

// NETWORK 49
//   PS6: IO : | AT %IX1.5
//   k6PressureLow: AT %MX619.5
k6PressureLow := NOT PS6;

// NETWORK 50

// NETWORK 51

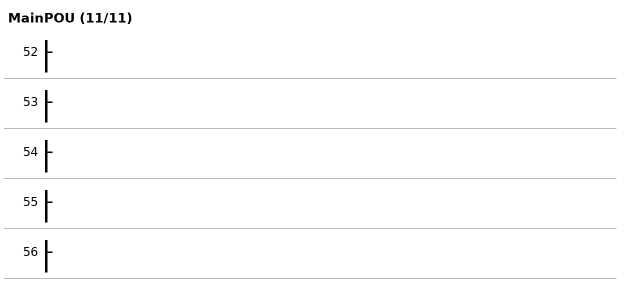
// NETWORK 52

// NETWORK 53

// NETWORK 54

// NETWORK 55

// NETWORK 56

END_PROGRAM

// MyController/Application/fx1
FUNCTION_BLOCK fx1
VAR_INPUT
	es: BOOL;
	tc: BOOL;
	setCycleTime: INT;
	setCylTime: INT;
	startCycle: BOOL;
	manOverride: BOOL;
END_VAR
VAR_OUTPUT
	elapsedTime: INT;
	cylOpenCmd: BOOL;
END_VAR
VAR
	setTimeMS: DINT;
	t1: TON;
	timeEN: BOOL;
	etDINT: DINT;
	t2: TP;
	t2EN: BOOL;
	cylOpenTime: TIME;
	
END_VAR

VAR RETAIN
	elapsedTimeMS: DINT;
	prevETMS: DINT;
END_VAR

setTimeMS := setCycleTime*1000;
etDINT := TIME_TO_DINT(t1.ET);
cylOpenTime := DINT_TO_TIME(setCylTime*1000);

t1(IN:= timeEN, PT:= T#999M);
t2(IN:= t2EN, PT:=cylOpenTime);

elapsedTime := DINT_TO_INT(elapsedTimeMS/1000);
elapsedTimeMS := prevETMS + etDINT;
cylOpenCmd := t2.Q;
IF startCycle THEN
IF es THEN
	IF tc OR manOverride THEN
		t2EN := FALSE;
		IF NOT cylOpenCmd THEN
			timeEN:= TRUE;
		END_IF
		
		IF elapsedTimeMS >= setTimeMS THEN
			t2EN := TRUE;
			timeEN := FALSE;
			prevETMS := 0;
		END_IF
	ELSE
		timeEN := FALSE;
		t2EN := FALSE;
		prevETMS := elapsedTimeMS;
	END_IF
ELSE
	timeEN := FALSE;
	t2EN := FALSE;
	prevETMS := elapsedTimeMS;
END_IF
ELSE
	t2EN := FALSE;
	timeEN := FALSE;
	prevETMS := 0;
END_IF

END_FUNCTION_BLOCK

// MyController/Application/fx2
FUNCTION_BLOCK fx2
VAR_INPUT
	cylOpen: BOOL;
	cycleStart: BOOL;
	setCount: INT;
	setCloseCount: INT;
	reset: BOOL;
END_VAR
VAR_OUTPUT
	actCount: INT;
	closeTopCyl: BOOL;
	stopCycle: BOOL;
	countComplete: BOOL;
END_VAR
VAR
	ctrReset: BOOL;
	ctr2Reset: BOOL;

	t1: ton;
	t1en: BOOL;
	setCloseCountCal: INT;
END_VAR
VAR RETAIN
	ctr1: CTU;
	ctr2: CTU;
	rtrig1: R_TRIG;
END_VAR

rtrig1(CLK:=cycleStart);
ctr1(CU:= cylOpen, RESET:= ctrReset, PV:= INT_TO_WORD(setCount));
ctr2(CU:= ctr1.Q, RESET:= ctr2Reset, PV:=1);
actCount := WORD_TO_INT(ctr1.CV);
setCloseCountCal := setCount - setCloseCount;
IF ctr1.Q THEN 
	countComplete := TRUE;
	stopCycle := TRUE;
ELSE
	stopCycle := FALSE;
END_IF

IF rtrig1.Q THEN
	ctrReset := TRUE;
	countComplete := FALSE;
	closeTopCyl := FALSE;
ELSE
	ctrReset := FALSE;
END_IF
t1(IN:= t1en, pt:= T#2S);	
IF ctr2.Q THEN
	IF actCount >= setCloseCountCal AND actcount < setCount THEN
		t1en:= TRUE;
		IF t1.Q THEN
			closeTopCyl := TRUE;
		END_IF
	ELSE
		closeTopCyl := FALSE;
		t1en:= FALSE;
	END_IF
	IF ctr2.CV = 2 THEN
		ctr2Reset := TRUE;
	END_IF
	IF setcount = 0 AND ctr2.CV = 2 THEN
		closetopcyl := TRUE;
	END_IF
	IF countComplete THEN
		closeTopCyl := FALSE;
	ELSE
		ctr2Reset := FALSE;
	END_IF
ELSE
	ctr2Reset := FALSE;
END_IF 
IF reset THEN
	ctrReset:= TRUE;
	ctr2Reset:=TRUE;
	closeTopCyl:=FALSE;
	stopCycle:=TRUE;
	countComplete:=FALSE;
	t1en:=FALSE;
END_IF

END_FUNCTION_BLOCK

// MyController/Application/CylOpenClose
FUNCTION_BLOCK CylOpenClose
VAR_INPUT
	manOpen: BOOL;
	AutoCmd: BOOL;
	manClose: BOOL;
END_VAR
VAR_OUTPUT
	out: BOOL;
END_VAR
VAR
	ftrig1: F_TRIG;
END_VAR

IF manOpen OR AutoCmd THEN
	out := TRUE;
END_IF
ftrig1(CLK:= AutoCmd);
IF manClose OR fTrig1.Q THEN
	out := FALSE;
END_IF

END_FUNCTION_BLOCK

// MyController/Application/HiddenPOU
FUNCTION HiddenPOU : BOOL

VAR_INPUT
	pHiddenFunc: POINTER TO WORD;
END_VAR
VAR
	pRead: POINTER TO BYTE;
	pWrite: POINTER TO BYTE;
END_VAR

pRead := pHiddenFunc + 400;
pWrite := pHiddenFunc + 4400;
HiddenPOU := TRUE;

END_FUNCTION
